# EPICS substitutions: gigeApp/Db/pluginTIFF.substitutions
#
# pluginTIFF.substitutions
#

file NDPluginBase.template
{
	{
	P=$(CAM):,
	R=TIFF$(N):,
	PORT=TIFF$(N),
	ADDR=0,
	TIMEOUT=1,
	NDARRAY_PORT=$(PLUGIN_SRC),
	NDARRAY_ADDR=0
	}
}

file NDFile.template
{
	{
	P=$(CAM):,
	R=TIFF$(N):,
	PORT=TIFF$(N),
	ADDR=0,
	TIMEOUT=1
	}
}

file NDFileTIFF.template
{
	{
	P=$(CAM):,
	R=TIFF$(N):,
	PORT=TIFF$(N),
	ADDR=0,
	TIMEOUT=1
	}
}
